PROGRAM P_SaveCurrentLanguage
VAR
END_VAR

RVL.currLanguage := VisuElems.CurrentLanguage;

MAIN.M_Log(reqLevel:=CVL.INFO, objectName:= 'P_SaveCurrentLanguage', sMsg:=RVL.currLanguage, errNo:= 0);

END_PROGRAM

(* stored: Version 1.1.0.1, ProductVersion 3.1.4024.3
   POU P_SaveCurrentLanguage: Id {cd5ba2db-3ead-47b2-8616-e429a147a88c}, SpecialFunc None *)
